FUNCTION_BLOCK FB_Tracklist IMPLEMENTS ITrackList
VAR_INPUT
END_VAR
VAR_OUTPUT
END_VAR
VAR
	_list : ARRAY [1..iMaxNumbMovers] OF ST_MoverData;
	_sorted : ARRAY [1..iMaxNumbMovers] OF ST_MoverData;
	_temp : ST_MoverData;
	i,j : INT;
END_VAR

METHOD AddMover : BOOL
VAR_INPUT
	data	: ST_MoverData;
END_VAR
VAR
	temp	: INT;
END_VAR
_list[data.id] := data;
END_METHOD

METHOD Sort : BOOL
// Step 1: Copy the list
_sorted := _list;

// Step 2: Bubble Sort the list
FOR i := 1 TO iMaxNumbMovers - 1 DO
    FOR j := i + 1 TO iMaxNumbMovers DO
        IF _sorted[i].pos > _sorted[j].pos THEN
            _temp := _sorted[i];
            _sorted[i] := _sorted[j];
            _sorted[j] := _temp;
        END_IF
    END_FOR
END_FOR
END_METHOD

END_FUNCTION_BLOCK

(* stored: Version 1.1.0.1, ProductVersion 3.1.4026.12
   POU FB_Tracklist: Id {546a42d1-a9e5-46d3-b826-00988018d01d}, SpecialFunc None
   Method AddMover: Id {19bcc54b-d09d-4767-9281-dabe045635c5}
   Method Sort: Id {5182b790-329f-48c5-abac-59d6da2e6290} *)
